Staubli VAL3: onF5Event.pgx

program onF5Event()
  local string l_sPage
  local string l_sItem
begin
  // look if the bButton is enable
  if bButton[4]
    // LOAD THE CYCLE PAGE
    l_sPage="kernel/page/production"
    call loadPage(l_sPage,l_sItem)
    //
    logMsg("[KERNEL] INTERFACE:PAGE Home Page")
    //
  endIf
end
